///////////
// Structure For Bousquet. Main Operating Data to be saved (ex: OPC).  
//////////

TYPE CB_AuxMVCB_Sch :
STRUCT
	//DI
	MesData					: CB ;      (* Object*)
	MesFuseBurned		    : BOOL ; 	(* The Fuse is burned*)
	MesEarth				: BOOL ; 	(* The Cell is grounded*)

END_STRUCT
END_TYPE

(* stored: Version 1.1.0.1, ProductVersion 3.1.4024.9
   DUT CB_AuxMVCB_Sch: Id {6050026c-f65b-4add-9d80-b4860ab1d6c0} *)
